// TIA Portal V18 export
DATA_BLOCK "ST10_StopperCtrl_DB"   // DB2601
// stored: AutoNumber false, InstanceOfName ST10_StopperCtrl, InstanceOfType FB
"ST10_StopperCtrl"
   // VAR
   //    Stopper { S7_SetPoint := 'True'} : Array[1..100] of "StopperCtrl";
   // END_VAR
BEGIN
END_DATA_BLOCK
